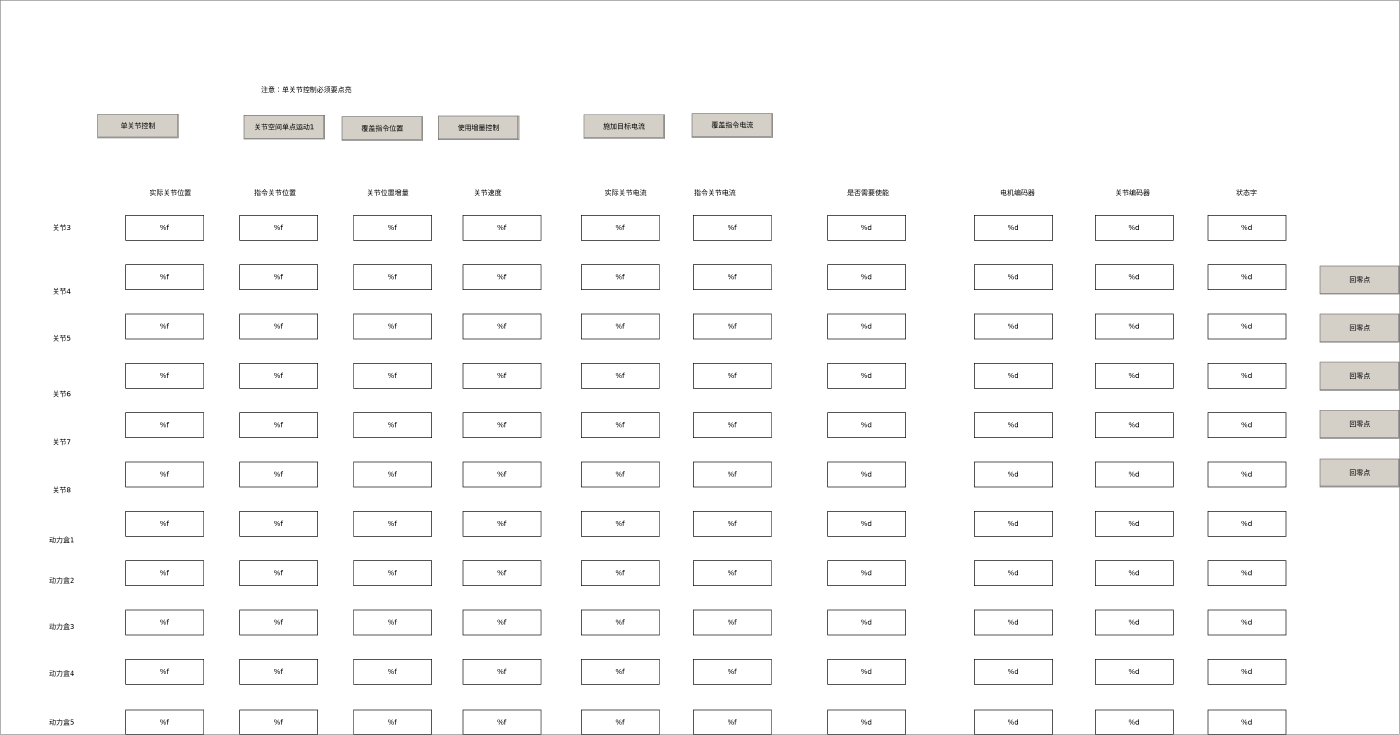
VISUALIZATION motion_a3  // 2212x1162
    Button (385,182 128x38), "关节空间单点运动1", colour toggle: g_motionTest.m_uiArmMode[3,1]
        tap g_motionTest.m_uiArmMode[3,1]
    Label (362,291 145x28), "指令关节位置"
    Label (194,290 150x30), "实际关节位置"
    Label (540,291 145x28), "关节位置增量"
    Label (698,291 145x28), "关节速度"
    Label (916,291 145x28), "实际关节电流"
    Label (1057,291 145x28), "指令关节电流"
    Rectangle (198,574 124x40), "%f", text variable: g_motionTest.m_actJntPos[3][1]
    Label (25,346 145x28), "关节3"
    Label (25,447 145x28), "关节4"
    Label (25,521 145x28), "关节5"
    Label (25,609 145x28), "关节6"
    Label (25,685 145x28), "关节7"
    Label (25,761 145x28), "关节8"
    Label (25,840 145x28), "动力盒1"
    Label (25,904 145x28), "动力盒2"
    Label (25,1128 145x28), "动力盒5"
    Label (25,977 145x28), "动力盒3"
    Label (25,1051 145x28), "动力盒4"
    Rectangle (198,652 124x40), "%f", text variable: g_motionTest.m_actJntPos[3][2]
    Rectangle (198,730 124x40), "%f", text variable: g_motionTest.m_actJntPos[3][3]
    Rectangle (198,808 124x40), "%f", text variable: g_motionTest.m_actJntPos[3][4]
    Rectangle (198,886 124x40), "%f", text variable: g_motionTest.m_actJntPos[3][5]
    Rectangle (198,964 124x40), "%f", text variable: g_motionTest.m_actJntPos[3][6]
    Rectangle (198,1042 124x40), "%f", text variable: g_motionTest.m_actJntPos[3][7]
    Rectangle (198,1122 124x40), "%f", text variable: g_motionTest.m_actJntPos[3][8]
    Rectangle (198,340 124x40), "%f", text variable: g_motionTest.m_actJntPosSetup[3][3]
    Rectangle (198,418 124x40), "%f", text variable: g_motionTest.m_actJntPosSetup[3][4]
    Rectangle (198,496 124x40), "%f", text variable: g_motionTest.m_actJntPosSetup[3][5]
    Rectangle (378,340 124x40), "%f", text variable: g_motionTest.m_targetJntPosSetup[3][3]
        OnMouseClick: write the text variable via Default
    Rectangle (378,418 124x40), "%f", text variable: g_motionTest.m_targetJntPosSetup[3][4]
        OnMouseClick: write the text variable via Default
    Rectangle (378,496 124x40), "%f", text variable: g_motionTest.m_targetJntPosSetup[3][5]
        OnMouseClick: write the text variable via Default
    Rectangle (378,574 124x40), "%f", text variable: g_motionTest.m_targetJntPosN8[3][1]
        OnMouseClick: write the text variable via Default
    Rectangle (378,652 124x40), "%f", text variable: g_motionTest.m_targetJntPosN8[3][2]
        OnMouseClick: write the text variable via Default
    Rectangle (378,730 124x40), "%f", text variable: g_motionTest.m_targetJntPosN8[3][3]
        OnMouseClick: write the text variable via Default
    Rectangle (378,808 124x40), "%f", text variable: g_motionTest.m_targetJntPosN8[3][4]
        OnMouseClick: write the text variable via Default
    Rectangle (378,886 124x40), "%f", text variable: g_motionTest.m_targetJntPosN8[3][5]
        OnMouseClick: write the text variable via Default
    Rectangle (378,964 124x40), "%f", text variable: g_motionTest.m_targetJntPosN8[3][6]
        OnMouseClick: write the text variable via Default
    Rectangle (378,1042 124x40), "%f", text variable: g_motionTest.m_targetJntPosN8[3][7]
        OnMouseClick: write the text variable via Default
    Rectangle (378,1122 124x40), "%f", text variable: g_motionTest.m_targetJntPosN8[3][8]
        OnMouseClick: write the text variable via Default
    Rectangle (558,340 124x40), "%f", text variable: g_motionTest.m_targetJntPosIncSetup[3][3]
        OnMouseClick: write the text variable via Default
    Rectangle (558,418 124x40), "%f", text variable: g_motionTest.m_targetJntPosIncSetup[3][4]
        OnMouseClick: write the text variable via Default
    Rectangle (558,496 124x40), "%f", text variable: g_motionTest.m_targetJntPosIncSetup[3][5]
        OnMouseClick: write the text variable via Default
    Rectangle (558,574 124x40), "%f", text variable: g_motionTest.m_targetJntPosIncN8[3][1]
        OnMouseClick: write the text variable via Default
    Rectangle (558,652 124x40), "%f", text variable: g_motionTest.m_targetJntPosIncN8[3][2]
        OnMouseClick: write the text variable via Default
    Rectangle (558,730 124x40), "%f", text variable: g_motionTest.m_targetJntPosIncN8[3][3]
        OnMouseClick: write the text variable via Default
    Rectangle (558,808 124x40), "%f", text variable: g_motionTest.m_targetJntPosIncN8[3][4]
        OnMouseClick: write the text variable via Default
    Rectangle (558,886 124x40), "%f", text variable: g_motionTest.m_targetJntPosIncN8[3][5]
        OnMouseClick: write the text variable via Default
    Rectangle (558,964 124x40), "%f", text variable: g_motionTest.m_targetJntPosIncN8[3][6]
        OnMouseClick: write the text variable via Default
    Rectangle (558,1042 124x40), "%f", text variable: g_motionTest.m_targetJntPosIncN8[3][7]
        OnMouseClick: write the text variable via Default
    Rectangle (558,1122 124x40), "%f", text variable: g_motionTest.m_targetJntPosIncN8[3][8]
        OnMouseClick: write the text variable via Default
    Rectangle (731,340 124x40), "%f", text variable: g_motionTest.m_targetJntVelSetup[3][3]
        OnMouseClick: write the text variable via Default
    Rectangle (731,418 124x40), "%f", text variable: g_motionTest.m_targetJntVelSetup[3][4]
        OnMouseClick: write the text variable via Default
    Rectangle (731,496 124x40), "%f", text variable: g_motionTest.m_targetJntVelSetup[3][5]
        OnMouseClick: write the text variable via Default
    Rectangle (731,574 124x40), "%f", text variable: g_motionTest.m_targetJntVel[3][1]
        OnMouseClick: write the text variable via Default
    Rectangle (731,652 124x40), "%f", text variable: g_motionTest.m_targetJntVel[3][2]
        OnMouseClick: write the text variable via Default
    Rectangle (731,730 124x40), "%f", text variable: g_motionTest.m_targetJntVel[3][3]
        OnMouseClick: write the text variable via Default
    Rectangle (731,808 124x40), "%f", text variable: g_motionTest.m_targetJntVel[3][4]
        OnMouseClick: write the text variable via Default
    Rectangle (731,886 124x40), "%f", text variable: g_motionTest.m_targetJntVel[3][5]
        OnMouseClick: write the text variable via Default
    Rectangle (731,964 124x40), "%f", text variable: g_motionTest.m_targetJntVel[3][6]
        OnMouseClick: write the text variable via Default
    Rectangle (731,1042 124x40), "%f", text variable: g_motionTest.m_targetJntVel[3][7]
        OnMouseClick: write the text variable via Default
    Rectangle (731,1122 124x40), "%f", text variable: g_motionTest.m_targetJntVel[3][8]
        OnMouseClick: write the text variable via Default
    Rectangle (918,340 124x40), "%f", text variable: g_motionTest.m_actJntCurrentSetup[3][3]
    Rectangle (918,418 124x40), "%f", text variable: g_motionTest.m_actJntCurrentSetup[3][4]
    Rectangle (918,496 124x40), "%f", text variable: g_motionTest.m_actJntCurrentSetup[3][5]
    Rectangle (918,574 124x40), "%f", text variable: g_motionTest.m_actJntCurrent[3][1]
    Rectangle (918,652 124x40), "%f", text variable: g_motionTest.m_actJntCurrent[3][2]
    Rectangle (918,730 124x40), "%f", text variable: g_motionTest.m_actJntCurrent[3][3]
    Rectangle (918,808 124x40), "%f", text variable: g_motionTest.m_actJntCurrent[3][4]
    Rectangle (918,886 124x40), "%f", text variable: g_motionTest.m_actJntCurrent[3][5]
    Rectangle (918,964 124x40), "%f", text variable: g_motionTest.m_actJntCurrent[3][6]
    Rectangle (918,1042 124x40), "%f", text variable: g_motionTest.m_actJntCurrent[3][7]
    Rectangle (918,1122 124x40), "%f", text variable: g_motionTest.m_actJntCurrent[3][8]
    Rectangle (1095,340 124x40), "%f", text variable: g_motionTest.m_targetJntCurrentSetup[3][3]
        OnMouseClick: write the text variable via Default
    Rectangle (1095,418 124x40), "%f", text variable: g_motionTest.m_targetJntCurrentSetup[3][4]
        OnMouseClick: write the text variable via Default
    Rectangle (1095,496 124x40), "%f", text variable: g_motionTest.m_targetJntCurrentSetup[3][5]
        OnMouseClick: write the text variable via Default
    Rectangle (1095,574 124x40), "%f", text variable: g_motionTest.m_targetJntCurrentN8[3][1]
        OnMouseClick: write the text variable via Default
    Rectangle (1095,652 124x40), "%f", text variable: g_motionTest.m_targetJntCurrentN8[3][2]
        OnMouseClick: write the text variable via Default
    Rectangle (1095,730 124x40), "%f", text variable: g_motionTest.m_targetJntCurrentN8[3][3]
        OnMouseClick: write the text variable via Default
    Rectangle (1095,808 124x40), "%f", text variable: g_motionTest.m_targetJntCurrentN8[3][4]
        OnMouseClick: write the text variable via Default
    Rectangle (1095,886 124x40), "%f", text variable: g_motionTest.m_targetJntCurrentN8[3][5]
        OnMouseClick: write the text variable via Default
    Rectangle (1095,964 124x40), "%f", text variable: g_motionTest.m_targetJntCurrentN8[3][6]
        OnMouseClick: write the text variable via Default
    Rectangle (1095,1042 124x40), "%f", text variable: g_motionTest.m_targetJntCurrentN8[3][7]
        OnMouseClick: write the text variable via Default
    Rectangle (1095,1122 124x40), "%f", text variable: g_motionTest.m_targetJntCurrentN8[3][8]
        OnMouseClick: write the text variable via Default
    Button (692,183 128x38), "使用增量控制", colour toggle: g_motionTest.m_singleMotorIncControl[3]
        toggle g_motionTest.m_singleMotorIncControl[3]
    Button (922,181 128x38), "施加目标电流", colour toggle: g_motionTest.m_uiArmMode[3,9]
        toggle g_motionTest.m_uiArmMode[3,9]
    Button (154,180 128x38), "单关节控制", colour toggle: g_motionTest.m_singleMotorControl[3]
        toggle g_motionTest.m_singleMotorControl[3] p2164770859=TRUE
    Label (374,127 220x30), "注意：单关节控制必须要点亮"
    Label (1299,290 145x30), "是否需要使能"
    Rectangle (1307,340 124x40), "%d", text variable: g_motionTest.m_jntEnableSetup[3][3]
        OnMouseClick: write the text variable via Default
    Rectangle (1307,418 124x40), "%d", text variable: g_motionTest.m_jntEnableSetup[3][4]
        OnMouseClick: write the text variable via Default
    Rectangle (1307,496 124x40), "%d", text variable: g_motionTest.m_jntEnableSetup[3][5]
        OnMouseClick: write the text variable via Default
    Rectangle (1307,574 124x40), "%d", text variable: g_motionTest.m_jntEnable[3][1]
        OnMouseClick: write the text variable via Default
    Rectangle (1307,652 124x40), "%d", text variable: g_motionTest.m_jntEnable[3][2]
        OnMouseClick: write the text variable via Default
    Label (1535,291 145x28), "电机编码器"
    Label (1717,291 145x28), "关节编码器"
    Label (1897,291 145x28), "状态字"
    Rectangle (1539,340 124x40), "%d", text variable: g_systemInfo.m_setupJntInfo[3,3].m_motorInput.m_motorEncoder
    Rectangle (1539,418 124x40), "%d", text variable: g_systemInfo.m_setupJntInfo[3,4].m_motorInput.m_motorEncoder
    Rectangle (1539,496 124x40), "%d", text variable: g_systemInfo.m_setupJntInfo[3,5].m_motorInput.m_motorEncoder
    Rectangle (1539,574 124x40), "%d", text variable: g_systemInfo.m_slaveJntInfo[3,1].m_motorInput.m_motorEncoder
    Rectangle (1539,652 124x40), "%d", text variable: g_systemInfo.m_slaveJntInfo[3,2].m_motorInput.m_motorEncoder
    Rectangle (1730,340 124x40), "%d", text variable: g_systemInfo.m_setupJntInfo[3,3].m_motorInput.m_linkEncoder
    Rectangle (1730,418 124x40), "%d", text variable: g_systemInfo.m_setupJntInfo[3,4].m_motorInput.m_linkEncoder
    Rectangle (1730,496 124x40), "%d", text variable: g_systemInfo.m_setupJntInfo[3,5].m_motorInput.m_linkEncoder
    Rectangle (1730,574 124x40), "%d", text variable: g_systemInfo.m_slaveJntInfo[3,1].m_motorInput.m_linkEncoder
    Rectangle (1730,652 124x40), "%d", text variable: g_systemInfo.m_slaveJntInfo[3,2].m_motorInput.m_linkEncoder
    Rectangle (1908,340 124x40), "%d", text variable: g_systemInfo.m_setupJntInfo[3,3].m_motorInput.m_statusWord
    Rectangle (1908,418 124x40), "%d", text variable: g_systemInfo.m_setupJntInfo[3,4].m_motorInput.m_statusWord
    Rectangle (1908,496 124x40), "%d", text variable: g_systemInfo.m_setupJntInfo[3,5].m_motorInput.m_statusWord
    Rectangle (1908,574 124x40), "%d", text variable: g_systemInfo.m_slaveJntInfo[3,1].m_motorInput.m_statusWord
    Rectangle (1908,652 124x40), "%d", text variable: g_systemInfo.m_slaveJntInfo[3,2].m_motorInput.m_statusWord
    Rectangle (1539,730 124x40), "%d", text variable: g_systemInfo.m_slaveJntInfo[3,3].m_motorInput.m_motorEncoder
    Rectangle (1539,808 124x40), "%d", text variable: g_systemInfo.m_slaveJntInfo[3,4].m_motorInput.m_motorEncoder
    Rectangle (1539,886 124x40), "%d", text variable: g_systemInfo.m_slaveJntInfo[3,5].m_motorInput.m_motorEncoder
    Rectangle (1539,964 124x40), "%d", text variable: g_systemInfo.m_slaveJntInfo[3,6].m_motorInput.m_motorEncoder
    Rectangle (1539,1042 124x40), "%d", text variable: g_systemInfo.m_slaveJntInfo[3,7].m_motorInput.m_motorEncoder
    Rectangle (1539,1122 124x40), "%d", text variable: g_systemInfo.m_slaveJntInfo[3,8].m_motorInput.m_motorEncoder
    Rectangle (1730,730 124x40), "%d", text variable: g_systemInfo.m_slaveJntInfo[3,3].m_motorInput.m_linkEncoder
    Rectangle (1730,808 124x40), "%d", text variable: g_systemInfo.m_slaveJntInfo[3,4].m_motorInput.m_linkEncoder
    Rectangle (1730,886 124x40), "%d", text variable: g_systemInfo.m_slaveJntInfo[3,5].m_motorInput.m_linkEncoder
    Rectangle (1730,964 124x40), "%d", text variable: g_systemInfo.m_slaveJntInfo[3,6].m_motorInput.m_linkEncoder
    Rectangle (1730,1042 124x40), "%d", text variable: g_systemInfo.m_slaveJntInfo[3,7].m_motorInput.m_linkEncoder
    Rectangle (1730,1122 124x40), "%d", text variable: g_systemInfo.m_slaveJntInfo[3,8].m_motorInput.m_linkEncoder
    Rectangle (1908,730 124x40), "%d", text variable: g_systemInfo.m_slaveJntInfo[3,3].m_motorInput.m_statusWord
    Rectangle (1908,808 124x40), "%d", text variable: g_systemInfo.m_slaveJntInfo[3,4].m_motorInput.m_statusWord
    Rectangle (1908,886 124x40), "%d", text variable: g_systemInfo.m_slaveJntInfo[3,5].m_motorInput.m_statusWord
    Rectangle (1908,964 124x40), "%d", text variable: g_systemInfo.m_slaveJntInfo[3,6].m_motorInput.m_statusWord
    Rectangle (1908,1042 124x40), "%d", text variable: g_systemInfo.m_slaveJntInfo[3,7].m_motorInput.m_statusWord
    Rectangle (1908,1122 124x40), "%d", text variable: g_systemInfo.m_slaveJntInfo[3,8].m_motorInput.m_statusWord
    Rectangle (1307,730 124x40), "%d", text variable: g_motionTest.m_jntEnable[3][3]
        OnMouseClick: write the text variable via Default
    Rectangle (1307,808 124x40), "%d", text variable: g_motionTest.m_jntEnable[3][4]
        OnMouseClick: write the text variable via Default
    Rectangle (1307,886 124x40), "%d", text variable: g_motionTest.m_jntEnable[3][5]
        OnMouseClick: write the text variable via Default
    Rectangle (1307,964 124x40), "%d", text variable: g_motionTest.m_jntEnable[3][6]
        OnMouseClick: write the text variable via Default
    Rectangle (1307,1042 124x40), "%d", text variable: g_motionTest.m_jntEnable[3][7]
        OnMouseClick: write the text variable via Default
    Rectangle (1307,1122 124x40), "%d", text variable: g_motionTest.m_jntEnable[3][8]
        OnMouseClick: write the text variable via Default
    Button (540,184 128x38), "覆盖指令位置", colour toggle: g_motionTest.m_coverCmdPos[3]
        tap g_motionTest.m_coverCmdPos[3]
    Button (2085,420 127x45), "回零点", colour toggle: g_motionTest.m_goHomeSetup[3][4]
        tap g_motionTest.m_goHomeSetup[3][4]
    Button (2085,496 127x45), "回零点", colour toggle: g_motionTest.m_goHomeSetup[3][5]
        tap g_motionTest.m_goHomeSetup[3][5]
    Button (2085,572 127x45), "回零点", colour toggle: g_motionTest.m_goHome[3][1]
        tap g_motionTest.m_goHome[3][1]
    Button (2085,648 127x45), "回零点", colour toggle: g_motionTest.m_goHome[3][2]
        tap g_motionTest.m_goHome[3][2]
    Button (2085,725 127x45), "回零点", colour toggle: g_motionTest.m_goHome[3][3]
        tap g_motionTest.m_goHome[3][3]
    Button (1093,179 128x38), "覆盖指令电流", colour toggle: g_motionTest.m_coverCmdCurrent[3]
        tap g_motionTest.m_coverCmdCurrent[3]
END_VISUALIZATION

(* stored: Version 1.1.0.1, ProductVersion 3.1.4024.11
   Visu motion_a3: Id {9de14b38-5aa0-4220-a0af-7cb06618bfb1} *)
